METHOD containsNo
VAR_INPUT
	(* current string to check *)
	stringToCheck	:ANY_STRING;
	(* string that must not be found in ``stringToCheck`` *)
	searchString	:ANY_STRING;
	(* ``TRUE`` means ignore cases; ``FALSE`` means cases must be equal too *)
	ignoreCases		:BOOL;
	(* message if the assertion is false *)
	message			:AssertMessage;
END_VAR
IF (stringToCheck.TypeClass <> searchString.TypeClass) THEN
	THIS^.assertionWasWrong(message, THIS^.getDebugInfo('containsNo'));
	RETURN;
END_IF

IF (stringToCheck.TypeClass = __SYSTEM.TYPE_CLASS.TYPE_STRING) THEN
	THIS^.win1252Assertions.win1252ContainsNo(
		stringToCheck := stringToCheck.pValue,
		searchString := searchString.pValue,
		ignoreCases := ignoreCases,
		message := message
	);
ELSIF (stringToCheck.TypeClass = __SYSTEM.TYPE_CLASS.TYPE_WSTRING) THEN
	THIS^.utf16Assertions.utf16ContainsNo(
		stringToCheck := stringToCheck.pValue,
		searchString := searchString.pValue,
		ignoreCases := ignoreCases,
		message := message
	);
END_IF
END_METHOD

(*

short summary
=================
This assertion method checks if the current string ``stringToCheck`` ends with ``end``

.. attention:: 
	All strings are handled as null terminated byte/word streams.
	For windows-1252 is end of the string 16#00
	For UTF-16 is end of the string 16#00_00

.. attention:: 
	Method uses ``ANY_STRING`` and for this it's not possible
	to use literals/constants, because for ``ANY`` types the
	compiler generates``__SYSTEM.AnyType`` and 
	``__SYSTEM.AnyType`` contains a pointer  

.. attention:: 
	end of the string is **ALWAYS** the right side of the string 
	even for writings which written from right to left like Hebrew or Arabic

.. <legal notes>

legal notes
=================
| SPDX-FileCopyrightText: © 2022 ekvip automation GmbH <info@ekvip.de>
| SPDX-License-Identifier: Apache-2.0
| For details check: Apache-2.0_

.. _Apache-2.0: https://www.apache.org/licenses/LICENSE-2.0

.. </legal notes>

parameters
=================

*)

METHOD endsWith
VAR_INPUT
	(* current string to check *)
	stringToCheck	:ANY_STRING;
	(* expected end of ``stringToCheck`` *)
	end				:ANY_STRING;
	(* ``TRUE`` means ignore cases; ``FALSE`` means cases must be equal too *)
	ignoreCases		:BOOL;
	(* ``TRUE`` means truncation of spaces on the right side of ``stringToCheck``*)
	trim			:BOOL;
	(* message if the assertion is false *)
	message			:AssertMessage;
END_VAR
IF (stringToCheck.TypeClass <> end.TypeClass) THEN
	THIS^.assertionWasWrong(message, THIS^.getDebugInfo('endsWith'));
	RETURN;
END_IF

IF (stringToCheck.TypeClass = __SYSTEM.TYPE_CLASS.TYPE_STRING) THEN
	THIS^.win1252Assertions.win1252EndsWith(
		stringToCheck := stringToCheck.pValue,
		end := end.pValue,
		ignoreCases := ignoreCases,
		trim := trim,
		message := message
	);
ELSIF (stringToCheck.TypeClass = __SYSTEM.TYPE_CLASS.TYPE_WSTRING) THEN
	THIS^.utf16Assertions.utf16EndsWith(
		stringToCheck := stringToCheck.pValue,
		end := end.pValue,
		ignoreCases := ignoreCases,
		trim := trim,
		message := message
	);	
END_IF
END_METHOD

(*

short summary
=================
This assertion method checks if the current string ``stringToCheck`` is empty

.. attention:: 
	All strings are handled as null terminated byte/word streams.
	For windows-1252 is end of the string 16#00
	For UTF-16 is end of the string 16#00_00

.. attention:: 
	Method uses ``ANY_STRING`` and for this it's not possible
	to use literals/constants, because for ``ANY`` types the
	compiler generates``__SYSTEM.AnyType`` and 
	``__SYSTEM.AnyType`` contains a pointer  

.. <legal notes>

legal notes
=================
| SPDX-FileCopyrightText: © 2022 ekvip automation GmbH <info@ekvip.de>
| SPDX-License-Identifier: Apache-2.0
| For details check: Apache-2.0_

.. _Apache-2.0: https://www.apache.org/licenses/LICENSE-2.0

.. </legal notes>

parameters
=================

*)

METHOD isEmpty
VAR_INPUT
	(* current string to check *)
	stringToCheck	:ANY_STRING;
	(* message if the assertion is false *)
	message			:AssertMessage;
END_VAR
VAR CONSTANT
	(* strings are null terminated *)
	END_OF_WINDOWS_1252_STRING	:BYTE := 16#00;
	(* strings are null terminated *)
	END_OF_UTF16_STRING	:WORD := 16#0000;
END_VAR
IF (stringToCheck.TypeClass = __SYSTEM.TYPE_CLASS.TYPE_STRING) THEN
	IF (stringToCheck.pValue^ <> END_OF_WINDOWS_1252_STRING) THEN
		THIS^.assertionWasWrong(message, THIS^.getDebugInfo('isEmpty'));
	END_IF
ELSIF (stringToCheck.TypeClass = __SYSTEM.TYPE_CLASS.TYPE_WSTRING) THEN
	IF (stringToCheck.pValue^ <> END_OF_UTF16_STRING) THEN
		THIS^.assertionWasWrong(message, THIS^.getDebugInfo('isEmpty'));
	END_IF
END_IF
END_METHOD

(*

short summary
=================
This assertion method checks if the current string ``stringToCheck`` is equal to ``expected``

.. attention:: 
	All strings are handled as null terminated byte/word streams.
	For windows-1252 is end of the string 16#00
	For UTF-16 is end of the string 16#00_00

.. attention:: 
	Method uses ``ANY_STRING`` and for this it's not possible
	to use literals/constants, because for ``ANY`` types the
	compiler generates``__SYSTEM.AnyType`` and 
	``__SYSTEM.AnyType`` contains a pointer  

.. <legal notes>

legal notes
=================
| SPDX-FileCopyrightText: © 2022 ekvip automation GmbH <info@ekvip.de>
| SPDX-License-Identifier: Apache-2.0
| For details check: Apache-2.0_

.. _Apache-2.0: https://www.apache.org/licenses/LICENSE-2.0

.. </legal notes>

parameters
=================

*)

METHOD isEqualTo
VAR_INPUT
	(* current string to check *)
	stringToCheck	:ANY_STRING;
	(* ``stringToCheck`` must be equal to expected *)
	expected		:ANY_STRING;
	(* ``TRUE`` means ignore cases; ``FALSE`` means cases must be equal too *)
	ignoreCases		:BOOL;
	(* message if the assertion is false *)
	message			:AssertMessage;
END_VAR
IF (stringToCheck.TypeClass <> expected.TypeClass) THEN
	THIS^.assertionWasWrong(message, THIS^.getDebugInfo('isEqualTo'));
	RETURN;
END_IF

IF (stringToCheck.TypeClass = __SYSTEM.TYPE_CLASS.TYPE_STRING) THEN
	THIS^.win1252Assertions.win1252IsEqualTo(
		stringToCheck := stringToCheck.pValue,
		expected := expected.pValue,
		ignoreCases := ignoreCases,
		message := message
	);
ELSIF (stringToCheck.TypeClass = __SYSTEM.TYPE_CLASS.TYPE_WSTRING) THEN
	THIS^.utf16Assertions.utf16IsEqualTo(
		stringToCheck := stringToCheck.pValue,
		expected := expected.pValue,
		ignoreCases := ignoreCases,
		message := message
	);	
END_IF
END_METHOD

(*

short summary
=================
This assertion method checks if the current string ``stringToCheck`` is not empty

.. attention:: 
	All strings are handled as null terminated byte/word streams.
	For windows-1252 is end of the string 16#00
	For UTF-16 is end of the string 16#00_00

.. attention:: 
	Method uses ``ANY_STRING`` and for this it's not possible
	to use literals/constants, because for ``ANY`` types the
	compiler generates``__SYSTEM.AnyType`` and 
	``__SYSTEM.AnyType`` contains a pointer  

.. <legal notes>

legal notes
=================
| SPDX-FileCopyrightText: © 2022 ekvip automation GmbH <info@ekvip.de>
| SPDX-License-Identifier: Apache-2.0
| For details check: Apache-2.0_

.. _Apache-2.0: https://www.apache.org/licenses/LICENSE-2.0

.. </legal notes>

parameters
=================

*)

METHOD isNotEmpty
VAR_INPUT
	(* current string to check *)
	stringToCheck	:ANY_STRING;
	(* message if the assertion is false *)
	message			:AssertMessage;
END_VAR
VAR CONSTANT
	(* strings are null terminated *)
	END_OF_WINDOWS_1252_STRING	:BYTE := 16#00;
	(* strings are null terminated *)
	END_OF_UTF16_STRING	:WORD := 16#0000;
END_VAR
IF (stringToCheck.TypeClass = __SYSTEM.TYPE_CLASS.TYPE_STRING) THEN
	IF (stringToCheck.pValue^ = END_OF_WINDOWS_1252_STRING) THEN
		THIS^.assertionWasWrong(message, THIS^.getDebugInfo('isNotEmpty'));
	END_IF
ELSIF (stringToCheck.TypeClass = __SYSTEM.TYPE_CLASS.TYPE_WSTRING) THEN
	IF (stringToCheck.pValue^ = END_OF_UTF16_STRING) THEN
		THIS^.assertionWasWrong(message, THIS^.getDebugInfo('isNotEmpty'));
	END_IF
END_IF
END_METHOD

(*

short summary
=================
This assertion method checks if the current string ``stringToCheck`` is not equal to ``unexpected``

.. attention:: 
	All strings are handled as null terminated byte/word streams.
	For windows-1252 is end of the string 16#00
	For UTF-16 is end of the string 16#00_00

.. attention:: 
	Method uses ``ANY_STRING`` and for this it's not possible
	to use literals/constants, because for ``ANY`` types the
	compiler generates``__SYSTEM.AnyType`` and 
	``__SYSTEM.AnyType`` contains a pointer  

.. <legal notes>

legal notes
=================
| SPDX-FileCopyrightText: © 2022 ekvip automation GmbH <info@ekvip.de>
| SPDX-License-Identifier: Apache-2.0
| For details check: Apache-2.0_

.. _Apache-2.0: https://www.apache.org/licenses/LICENSE-2.0

.. </legal notes>

parameters
=================

*)

METHOD isNotEqualTo
VAR_INPUT
	(* current string to check *)
	stringToCheck	:ANY_STRING;
	(* ``stringToCheck`` must be not equal to expected *)
	unexpected		:ANY_STRING;
	(* ``TRUE`` means ignore cases; ``FALSE`` means cases must be equal too *)
	ignoreCases		:BOOL;
	(* message if the assertion is false *)
	message			:AssertMessage;
END_VAR
IF (stringToCheck.TypeClass <> unexpected.TypeClass) THEN
	RETURN;
END_IF

IF (stringToCheck.TypeClass = __SYSTEM.TYPE_CLASS.TYPE_STRING) THEN
	THIS^.win1252Assertions.win1252IsNotEqualTo(
		stringToCheck := stringToCheck.pValue,
		unexpected := unexpected.pValue,
		ignoreCases := ignoreCases,
		message := message
	);
ELSIF (stringToCheck.TypeClass = __SYSTEM.TYPE_CLASS.TYPE_WSTRING) THEN
	THIS^.utf16Assertions.utf16IsNotEqualTo(
		stringToCheck := stringToCheck.pValue,
		unexpected := unexpected.pValue,
		ignoreCases := ignoreCases,
		message := message
	);	
END_IF
END_METHOD

(*

short summary
=================
This assertion method checks if the current string ``stringToCheck`` is length
is between ``minLenght`` and ``maxLenght``

.. attention:: 
	All strings are handled as null terminated byte/word streams.
	For windows-1252 is end of the string 16#00
	For UTF-16 is end of the string 16#00_00

.. attention:: 
	Method uses ``ANY_STRING`` and for this it's not possible
	to use literals/constants, because for ``ANY`` types the
	compiler generates``__SYSTEM.AnyType`` and 
	``__SYSTEM.AnyType`` contains a pointer  

.. <legal notes>

legal notes
=================
| SPDX-FileCopyrightText: © 2022 ekvip automation GmbH <info@ekvip.de>
| SPDX-License-Identifier: Apache-2.0
| For details check: Apache-2.0_

.. _Apache-2.0: https://www.apache.org/licenses/LICENSE-2.0

.. </legal notes>

parameters
=================

*)

METHOD lenghtIsBetween
VAR_INPUT
	(* current string to check *)
	stringToCheck	:ANY_STRING;
	(* lower limit of the string length *)
	minLenght		:UDINT;
	(* upper limit of the string length *)
	maxLenght		:UDINT;
	(* message if the assertion is false *)
	message			:AssertMessage;
END_VAR
IF (stringToCheck.TypeClass = __SYSTEM.TYPE_CLASS.TYPE_STRING) THEN
	THIS^.win1252Assertions.win1252LengthIsBetween(
		stringToCheck	:= stringToCheck.pValue,
		minLenght		:= minLenght,
		maxLenght		:= maxLenght,
		message			:= message
	);
ELSIF (stringToCheck.TypeClass = __SYSTEM.TYPE_CLASS.TYPE_WSTRING) THEN
	THIS^.utf16Assertions.utf16LengthIsBetween(
		stringToCheck	:= stringToCheck.pValue,
		minLenght		:= minLenght,
		maxLenght		:= maxLenght,
		message			:= message
	);	
END_IF
END_METHOD

(*

short summary
=================
This assertion method checks if the current string ``stringToCheck`` is length
is equal to ``expectedLength``

.. attention:: 
	All strings are handled as null terminated byte/word streams.
	For windows-1252 is end of the string 16#00
	For UTF-16 is end of the string 16#00_00

.. attention:: 
	Method uses ``ANY_STRING`` and for this it's not possible
	to use literals/constants, because for ``ANY`` types the
	compiler generates``__SYSTEM.AnyType`` and 
	``__SYSTEM.AnyType`` contains a pointer  

.. <legal notes>

legal notes
=================
| SPDX-FileCopyrightText: © 2022 ekvip automation GmbH <info@ekvip.de>
| SPDX-License-Identifier: Apache-2.0
| For details check: Apache-2.0_

.. _Apache-2.0: https://www.apache.org/licenses/LICENSE-2.0

.. </legal notes>

parameters
=================

*)

METHOD lenghtIsExact
VAR_INPUT
	(* current string to check *)
	stringToCheck	:ANY_STRING;
	(* expected length of ``stringToCheck`` *)
	expectedLength	:UDINT;
	(* message if the assertion is false *)
	message			:AssertMessage;
END_VAR
IF (stringToCheck.TypeClass = __SYSTEM.TYPE_CLASS.TYPE_STRING) THEN
	THIS^.win1252Assertions.win1252LenghtIsExact(
		stringToCheck	:= stringToCheck.pValue,
		expectedLength	:= expectedLength,
		message			:= message
	);
ELSIF (stringToCheck.TypeClass = __SYSTEM.TYPE_CLASS.TYPE_WSTRING) THEN
	THIS^.utf16Assertions.utf16LenghtIsExact(
		stringToCheck	:= stringToCheck.pValue,
		expectedLength	:= expectedLength,
		message			:= message
	);	
END_IF
END_METHOD

(*

short summary
=================
This assertion method checks if the current string ``stringToCheck`` is length
is equal or less than to ``maxLength``

.. attention:: 
	All strings are handled as null terminated byte/word streams.
	For windows-1252 is end of the string 16#00
	For UTF-16 is end of the string 16#00_00

.. attention:: 
	Method uses ``ANY_STRING`` and for this it's not possible
	to use literals/constants, because for ``ANY`` types the
	compiler generates``__SYSTEM.AnyType`` and 
	``__SYSTEM.AnyType`` contains a pointer  

.. <legal notes>

legal notes
=================
| SPDX-FileCopyrightText: © 2022 ekvip automation GmbH <info@ekvip.de>
| SPDX-License-Identifier: Apache-2.0
| For details check: Apache-2.0_

.. _Apache-2.0: https://www.apache.org/licenses/LICENSE-2.0

.. </legal notes>

parameters
=================

*)

METHOD lenghtIsMax
VAR_INPUT
	(* current string to check *)
	stringToCheck	:ANY_STRING;
	(* upper limit of the length of ``stringToCheck`` *)
	maxLength		:UDINT;
	(* message if the assertion is false *)
	message			:AssertMessage;
END_VAR
IF (stringToCheck.TypeClass = __SYSTEM.TYPE_CLASS.TYPE_STRING) THEN
	THIS^.win1252Assertions.win1252LenghtIsMax(
		stringToCheck	:= stringToCheck.pValue,
		maxLength		:= maxLength,
		message			:= message
	);
ELSIF (stringToCheck.TypeClass = __SYSTEM.TYPE_CLASS.TYPE_WSTRING) THEN
	THIS^.utf16Assertions.utf16LenghtIsMax(
		stringToCheck	:= stringToCheck.pValue,
		maxLength		:= maxLength,
		message			:= message
	);	
END_IF
END_METHOD

(*

short summary
=================
This assertion method checks if the current string ``stringToCheck`` is length
is equal or grater than to ``minLength``

.. attention:: 
	All strings are handled as null terminated byte/word streams.
	For windows-1252 is end of the string 16#00
	For UTF-16 is end of the string 16#00_00

.. attention:: 
	Method uses ``ANY_STRING`` and for this it's not possible
	to use literals/constants, because for ``ANY`` types the
	compiler generates``__SYSTEM.AnyType`` and 
	``__SYSTEM.AnyType`` contains a pointer  

.. <legal notes>

legal notes
=================
| SPDX-FileCopyrightText: © 2022 ekvip automation GmbH <info@ekvip.de>
| SPDX-License-Identifier: Apache-2.0
| For details check: Apache-2.0_

.. _Apache-2.0: https://www.apache.org/licenses/LICENSE-2.0

.. </legal notes>

parameters
=================

*)

METHOD lenghtIsMin
VAR_INPUT
	(* current string to check *)
	stringToCheck	:ANY_STRING;
	(* lower limit of the length of ``stringToCheck`` *)
	minLength		:UDINT;
	(* message if the assertion is false *)
	message			:AssertMessage;
END_VAR
IF (stringToCheck.TypeClass = __SYSTEM.TYPE_CLASS.TYPE_STRING) THEN
	THIS^.win1252Assertions.win1252LenghtIsMin(
		stringToCheck	:= stringToCheck.pValue,
		minLength		:= minLength,
		message			:= message
	);
ELSIF (stringToCheck.TypeClass = __SYSTEM.TYPE_CLASS.TYPE_WSTRING) THEN
	THIS^.utf16Assertions.utf16LenghtIsMin(
		stringToCheck	:= stringToCheck.pValue,
		minLength		:= minLength,
		message			:= message
	);
END_IF
END_METHOD

(*

short summary
=================
This methods is the setter for the callback class if an assertion was false

.. <legal notes>

legal notes
=================
| SPDX-FileCopyrightText: © 2022 ekvip automation GmbH <info@ekvip.de>
| SPDX-License-Identifier: Apache-2.0
| For details check: Apache-2.0_

.. _Apache-2.0: https://www.apache.org/licenses/LICENSE-2.0

.. </legal notes>

parameters
=================

*)

METHOD setCallBack
VAR_INPUT
	(* the class that must be informed if an assertion is false *)
	callBack	:IAssertCallback;  
END_VAR
SUPER^.setCallBack(callBack);
THIS^.win1252Assertions.setCallBack(callBack);
THIS^.utf16Assertions.setCallBack(callBack);
END_METHOD

(*

short summary
=================
This assertion method checks if the current string ``stringToCheck`` starts with ``start``

.. attention:: 
	All strings are handled as null terminated byte/word streams.
	For windows-1252 is end of the string 16#00
	For UTF-16 is end of the string 16#00_00

.. attention:: 
	Method uses ``ANY_STRING`` and for this it's not possible
	to use literals/constants, because for ``ANY`` types the
	compiler generates``__SYSTEM.AnyType`` and 
	``__SYSTEM.AnyType`` contains a pointer  

.. attention:: 
	start of the string is **ALWAYS** the left side of the string 
	even for writings which written from right to left like Hebrew or Arabic

.. <legal notes>

legal notes
=================
| SPDX-FileCopyrightText: © 2022 ekvip automation GmbH <info@ekvip.de>
| SPDX-License-Identifier: Apache-2.0
| For details check: Apache-2.0_

.. _Apache-2.0: https://www.apache.org/licenses/LICENSE-2.0

.. </legal notes>

parameters
=================

*)

METHOD startsWith
VAR_INPUT
	(* current string to check *)
	stringToCheck	:ANY_STRING;
	(* expected start of ``stringToCheck`` *)
	start			:ANY_STRING;
	(* ``TRUE`` means ignore cases; ``FALSE`` means cases must be equal too *)
	ignoreCases		:BOOL;
	(* ``TRUE`` means truncation of spaces on the left side of ``stringToCheck``*)
	trim			:BOOL;
	(* message if the assertion is false *)
	message			:AssertMessage;
END_VAR
IF (stringToCheck.TypeClass <> start.TypeClass) THEN
	THIS^.assertionWasWrong(message, THIS^.getDebugInfo('startsWith'));
	RETURN;
END_IF

IF (stringToCheck.TypeClass = __SYSTEM.TYPE_CLASS.TYPE_STRING) THEN
	THIS^.win1252Assertions.win1252StartsWith(
		stringToCheck := stringToCheck.pValue,
		start := start.pValue,
		ignoreCases := ignoreCases,
		trim := trim,
		message := message
	);
ELSIF (stringToCheck.TypeClass = __SYSTEM.TYPE_CLASS.TYPE_WSTRING) THEN
	THIS^.utf16Assertions.utf16StartsWith(
		stringToCheck := stringToCheck.pValue,
		start := start.pValue,
		ignoreCases := ignoreCases,
		trim := trim,
		message := message
	);
END_IF
END_METHOD

END_FUNCTION_BLOCK

// ---- Assertor/Assertions/TimeAssertions/classes/TimeAssertions.TcPOU
(*

short summary
=================
This class implements the interface :ref:`ITimeAssertions`.
It provides assertions for time data types
For ``LTIME`` assertions use :ref:`TimeAssertions.long`.
For ``TIME`` assertions use :ref:`TimeAssertions.simple`.


.. <legal notes>

legal notes
=================
| SPDX-FileCopyrightText: © 2022 ekvip automation GmbH <info@ekvip.de>
| SPDX-License-Identifier: Apache-2.0
| For details check: Apache-2.0_

.. _Apache-2.0: https://www.apache.org/licenses/LICENSE-2.0

.. </legal notes>

methods and properties
=========================

*)

{attribute 'reflection'}
FUNCTION_BLOCK INTERNAL TimeAssertions EXTENDS CNM_AbstractObject.Object IMPLEMENTS ITimeAssertions, IAssertCallBackSetter
VAR
	(* class to handle TIME assertions *)
	simpleTimeAssertions	:SimpleTimeAssertions();
	(* class to handle LTIME assertions *)
	longTimeAssertions		:LongTimeAssertions();
END_VAR

(*

short summary
=================
This abstract property returns the class name of the concrete object, 
It's for debugging purpose

.. <legal notes>

legal notes
=================
| SPDX-FileCopyrightText: © 2022 ekvip automation GmbH <info@ekvip.de>
| SPDX-License-Identifier: Apache-2.0
| For details check: Apache-2.0_

.. _Apache-2.0: https://www.apache.org/licenses/LICENSE-2.0

.. </legal notes>

*)

PROPERTY className :ClassName
GET
className := 'CNM_AssertionInterfaceLib.TimeAssertions';
END_GET
END_PROPERTY

(*

short summary
=================
Returns an interface (:ref:`I64BitTimeAssertions`)
with assert statements for 64 bit times 

.. <legal notes>

legal notes
=================
| SPDX-FileCopyrightText: © 2022 ekvip automation GmbH <info@ekvip.de>
| SPDX-License-Identifier: Apache-2.0
| For details check: Apache-2.0_

.. _Apache-2.0: https://www.apache.org/licenses/LICENSE-2.0

.. </legal notes>

*)

PROPERTY long :I64BitTimeAssertions
GET
long := THIS^.longTimeAssertions;
END_GET
END_PROPERTY

(*

short summary
=================
This methods is the setter for the callback class if an assertion was false

.. <legal notes>

legal notes
=================
| SPDX-FileCopyrightText: © 2022 ekvip automation GmbH <info@ekvip.de>
| SPDX-License-Identifier: Apache-2.0
| For details check: Apache-2.0_

.. _Apache-2.0: https://www.apache.org/licenses/LICENSE-2.0

.. </legal notes>

parameters
=================

*)

METHOD setCallBack
VAR_INPUT
	(* the class that must be informed if an assertion is false *)
	callBack	:IAssertCallback;  
END_VAR
THIS^.simpleTimeAssertions.setCallBack(callBack);
THIS^.longTimeAssertions.setCallBack(callBack);
END_METHOD

(*

short summary
=================
Returns an interface (:ref:`I32BitTimeAssertions`)
with assert statements for 32 bit times 

.. <legal notes>

legal notes
=================
| SPDX-FileCopyrightText: © 2022 ekvip automation GmbH <info@ekvip.de>
| SPDX-License-Identifier: Apache-2.0
| For details check: Apache-2.0_

.. _Apache-2.0: https://www.apache.org/licenses/LICENSE-2.0

.. </legal notes>

*)

PROPERTY simple :I32BitTimeAssertions
GET
simple := THIS^.simpleTimeAssertions;
END_GET
END_PROPERTY

END_FUNCTION_BLOCK

// ---- Assertor/Assertions/TimeAssertions/Time/classes/SimpleTimeAssertions.TcPOU
(*

short summary
=================
This class implements the interface :ref:`I32BitTimeAssertions`. 
It contains the assert statements for the data type ``TIME``

.. <legal notes>

legal notes
=================
| SPDX-FileCopyrightText: © 2022 ekvip automation GmbH <info@ekvip.de>
| SPDX-License-Identifier: Apache-2.0
| For details check: Apache-2.0_

.. _Apache-2.0: https://www.apache.org/licenses/LICENSE-2.0

.. </legal notes>

methods and properties
=========================

*)

{attribute 'reflection'}
FUNCTION_BLOCK INTERNAL SimpleTimeAssertions EXTENDS AbstactAssertion IMPLEMENTS I32BitTimeAssertions
VAR CONSTANT
	(* maximum value for the data type ``TIME`` *)
	MAX_TIME	:TIME := TO_TIME(16#FF_FF_FF_FF);
END_VAR

(*

short summary
=================
This abstract property returns the class name of the concrete object, 
It's for debugging purpose

.. <legal notes>

legal notes
=================
| SPDX-FileCopyrightText: © 2022 ekvip automation GmbH <info@ekvip.de>
| SPDX-License-Identifier: Apache-2.0
| For details check: Apache-2.0_

.. _Apache-2.0: https://www.apache.org/licenses/LICENSE-2.0

.. </legal notes>

*)

PROPERTY className :ClassName
GET
className := 'CNM_AssertionInterfaceLib.SimplyTimeAssertions';
END_GET
END_PROPERTY

(*

short summary
=================
This method returns the passed time since the timestamp was created

.. <legal notes>

legal notes
=================
| SPDX-FileCopyrightText: © 2022 ekvip automation GmbH <info@ekvip.de>
| SPDX-License-Identifier: Apache-2.0
| For details check: Apache-2.0_

.. _Apache-2.0: https://www.apache.org/licenses/LICENSE-2.0

.. </legal notes>

parameters
=================
:return: passed time since ``startTime``

*)

METHOD PROTECTED getTimePassed :TIME
VAR_INPUT
	(* timestamp start *)
	startTime	:TIME;
END_VAR
VAR
	(* current time to calculate the passed time *)
	currentTime	:TIME;
END_VAR
currentTime := TIME();
IF (currentTime > startTime) THEN
	getTimePassed := (currentTime - startTime);
ELSE
	getTimePassed := ((THIS^.MAX_TIME - startTime) + currentTime);
END_IF
END_METHOD

(*

short summary
=================
This assertion method checks whether time has elapsed since the timestamp time

.. <legal notes>

legal notes
=================
| SPDX-FileCopyrightText: © 2022 ekvip automation GmbH <info@ekvip.de>
| SPDX-License-Identifier: Apache-2.0
| For details check: Apache-2.0_

.. _Apache-2.0: https://www.apache.org/licenses/LICENSE-2.0

.. </legal notes>

parameters
=================

*)

METHOD timeHasExpired
VAR_INPUT
	(* start time you get it with ``TIME()`` *)
	timestamp		:TIME;
	(* timeout like ``t#300ms`` *)
	expiringTime	:TIME;
	(* message if the assertion is false *)
	message			:AssertMessage;
END_VAR
VAR
	(* measured passed time *)
	passedTime		:TIME;
END_VAR
passedTime := THIS^.getTimePassed(timestamp);
IF (passedTime < expiringTime) THEN
	THIS^.assertionWasWrong(
		message			:= message,
		additionalText	:= THIS^.getDebugInfo('timeHasExpired')
	);	
END_IF
END_METHOD

(*

short summary
=================
This assertion method checks that the time since the timestamp time has not yet elapsed

.. <legal notes>

legal notes
=================
| SPDX-FileCopyrightText: © 2022 ekvip automation GmbH <info@ekvip.de>
| SPDX-License-Identifier: Apache-2.0
| For details check: Apache-2.0_

.. _Apache-2.0: https://www.apache.org/licenses/LICENSE-2.0

.. </legal notes>

parameters
=================

*)

METHOD timeHasNotExpired
VAR_INPUT
	(* start time you get it with ``TIME()`` *)
	timestamp		:TIME;
	(* timeout like ``t#300ms`` *)
	expiringTime	:TIME;
	(* message if the assertion is false *)
	message			:AssertMessage;
END_VAR
VAR
	(* measured passed time *)
	passedTime		:TIME;
END_VAR
passedTime := THIS^.getTimePassed(timestamp);
IF (passedTime >= expiringTime) THEN
	THIS^.assertionWasWrong(
		message			:= message,
		additionalText	:= THIS^.getDebugInfo('timeHasNotExpired')
	);	
END_IF
END_METHOD

(*

short summary
=================
This assertion method checks if the current value is equal to the expected value

.. <legal notes>

legal notes
=================
| SPDX-FileCopyrightText: © 2022 ekvip automation GmbH <info@ekvip.de>
| SPDX-License-Identifier: Apache-2.0
| For details check: Apache-2.0_

.. _Apache-2.0: https://www.apache.org/licenses/LICENSE-2.0

.. </legal notes>

parameters
=================

*)

METHOD valueIsEqualTo
VAR_INPUT
	(* current value to check *)
	currentValue	:TIME;
	(* expected value to compare *)
	expectedValue	:TIME;
	(* message if the assertion is false *)
	message			:AssertMessage;
END_VAR
IF (currentValue <> expectedValue) THEN
	THIS^.assertionWasWrong(
		message			:= message,
		additionalText	:= THIS^.getDebugInfo('valueIsEqualTo')
	);	
END_IF
END_METHOD

(*

short summary
=================
This assertion method checks if the current value is greater than the less value

.. <legal notes>

legal notes
=================
| SPDX-FileCopyrightText: © 2022 ekvip automation GmbH <info@ekvip.de>
| SPDX-License-Identifier: Apache-2.0
| For details check: Apache-2.0_

.. _Apache-2.0: https://www.apache.org/licenses/LICENSE-2.0

.. </legal notes>

parameters
=================

*)

METHOD valueIsGreaterThan
VAR_INPUT
	(* current value to check *)
	currentValue	:TIME;
	(* less than lower limit *)
	lessValue		:TIME;
	(* message if the assertion is false *)
	message			:AssertMessage;
END_VAR
IF (currentValue <= lessValue) THEN
	THIS^.assertionWasWrong(
		message			:= message,
		additionalText	:= THIS^.getDebugInfo('valueIsGreaterThan')
	);	
END_IF
END_METHOD

(*

short summary
=================
This assertion method checks if the current value is inside a limit

.. attention:: 
	limits are included: ``valueIsInRangeOf(t#3ms,t#3ms ,t#3ms)`` is a true assertion

.. <legal notes>

legal notes
=================
| SPDX-FileCopyrightText: © 2022 ekvip automation GmbH <info@ekvip.de>
| SPDX-License-Identifier: Apache-2.0
| For details check: Apache-2.0_

.. _Apache-2.0: https://www.apache.org/licenses/LICENSE-2.0

.. </legal notes>

parameters
=================

*)

METHOD valueIsInRangeOf
VAR_INPUT
	(* lower limit for the current value *)
	lowerLimit		:TIME;
	(* current value to check *)
	currentValue	:TIME;
	(* upper limit for the current value *)
	upperLimit		:TIME;
	(* message if the assertion is false *)
	message			:AssertMessage;
END_VAR
IF ((currentValue < lowerLimit) OR (currentValue > upperLimit)) THEN
	THIS^.assertionWasWrong(
		message			:= message,
		additionalText	:= THIS^.getDebugInfo('valueIsInRangeOf')
	);	
END_IF
END_METHOD

(*

short summary
=================
This assertion method checks if the current value is less than the greater value

.. <legal notes>

legal notes
=================
| SPDX-FileCopyrightText: © 2022 ekvip automation GmbH <info@ekvip.de>
| SPDX-License-Identifier: Apache-2.0
| For details check: Apache-2.0_

.. _Apache-2.0: https://www.apache.org/licenses/LICENSE-2.0

.. </legal notes>

parameters
=================

*)

METHOD valueIsLessThan
VAR_INPUT
	(* current value to check *)
	currentValue	:TIME;
	(* greater than upper limit *)
	greaterValue	:TIME;
	(* message if the assertion is false *)
	message			:AssertMessage;
END_VAR
IF (currentValue >= greaterValue) THEN
	THIS^.assertionWasWrong(
		message			:= message,
		additionalText	:= THIS^.getDebugInfo('valueIsLessThan')
	);	
END_IF
END_METHOD

(*

short summary
=================
This assertion method checks if the current value is less than or equal to the maximum value

.. <legal notes>

legal notes
=================
| SPDX-FileCopyrightText: © 2022 ekvip automation GmbH <info@ekvip.de>
| SPDX-License-Identifier: Apache-2.0
| For details check: Apache-2.0_

.. _Apache-2.0: https://www.apache.org/licenses/LICENSE-2.0

.. </legal notes>

parameters
=================

*)

METHOD valueIsMax
VAR_INPUT
	(* current value to check *)
	currentValue	:TIME;
	(* upper limit for the current value *)
	maximumValue	:TIME;
	(* message if the assertion is false *)
	message			:AssertMessage;
END_VAR
IF (currentValue > maximumValue) THEN
	THIS^.assertionWasWrong(
		message			:= message,
		additionalText	:= THIS^.getDebugInfo('valueIsMax')
	);	
END_IF
END_METHOD

(*

short summary
=================
This assertion method checks if the current value is greater than or equal to the minimum value

.. <legal notes>

legal notes
=================
| SPDX-FileCopyrightText: © 2022 ekvip automation GmbH <info@ekvip.de>
| SPDX-License-Identifier: Apache-2.0
| For details check: Apache-2.0_

.. _Apache-2.0: https://www.apache.org/licenses/LICENSE-2.0

.. </legal notes>

parameters
=================

*)

METHOD valueIsMin
VAR_INPUT
	(* current value to check *)
	currentValue	:TIME;
	(* lower limit for the current value *)
	minimumValue	:TIME;
	(* message if the assertion is false *)
	message			:AssertMessage;
END_VAR
IF (currentValue < minimumValue) THEN
	THIS^.assertionWasWrong(
		message			:= message,
		additionalText	:= THIS^.getDebugInfo('valueIsMin')
	);	
END_IF
END_METHOD

(*

short summary
=================
This assertion method checks if the current value is not equal to the unexpected value

.. <legal notes>

legal notes
=================
| SPDX-FileCopyrightText: © 2022 ekvip automation GmbH <info@ekvip.de>
| SPDX-License-Identifier: Apache-2.0
| For details check: Apache-2.0_

.. _Apache-2.0: https://www.apache.org/licenses/LICENSE-2.0

.. </legal notes>

parameters
=================

*)

METHOD valueIsNotEqualTo
VAR_INPUT
	(* current value to check *)
	currentValue	:TIME;
	(* unexpected value to compare *)
	unexpectedValue	:TIME;
	(* message if the assertion is false *)
	message			:AssertMessage;
END_VAR
IF (currentValue = unexpectedValue) THEN
	THIS^.assertionWasWrong(
		message			:= message,
		additionalText	:= THIS^.getDebugInfo('valueIsNotEqualTo')
	);	
END_IF
END_METHOD

END_FUNCTION_BLOCK

// ---- Assertor/Assertions/TimeAssertions/LTime/classes/LongTimeAssertions.TcPOU
(*

short summary
=================
This class implements the interface :ref:`I64BitTimeAssertions`. 
It provides the assert statements for the data type ``LTIME``

.. <legal notes>

legal notes
=================
| SPDX-FileCopyrightText: © 2022 ekvip automation GmbH <info@ekvip.de>
| SPDX-License-Identifier: Apache-2.0
| For details check: Apache-2.0_

.. _Apache-2.0: https://www.apache.org/licenses/LICENSE-2.0

.. </legal notes>

methods and properties
=========================

*)

{attribute 'reflection'}
FUNCTION_BLOCK INTERNAL LongTimeAssertions EXTENDS AbstactAssertion IMPLEMENTS I64BitTimeAssertions
VAR CONSTANT
	(* maximum value for the data type ``LTIME`` *)
	MAX_TIME	:LTIME := TO_LTIME(16#FFFF_FFFF_FFFF_FFFF);
END_VAR

(*

short summary
=================
This abstract property returns the class name of the concrete object, 
It's for debugging purpose

.. <legal notes>

legal notes
=================
| SPDX-FileCopyrightText: © 2022 ekvip automation GmbH <info@ekvip.de>
| SPDX-License-Identifier: Apache-2.0
| For details check: Apache-2.0_

.. _Apache-2.0: https://www.apache.org/licenses/LICENSE-2.0

.. </legal notes>

*)

PROPERTY className :ClassName
GET
className := 'CNM_AssertionInterfaceLib.LongTimeAssertions';
END_GET
END_PROPERTY

(*

short summary
=================
This method returns the passed time since the timestamp was created

.. <legal notes>

legal notes
=================
| SPDX-FileCopyrightText: © 2022 ekvip automation GmbH <info@ekvip.de>
| SPDX-License-Identifier: Apache-2.0
| For details check: Apache-2.0_

.. _Apache-2.0: https://www.apache.org/licenses/LICENSE-2.0

.. </legal notes>

parameters
=================
:return: passed time since ``startTime``

*)

METHOD PROTECTED getTimePassed :LTIME
VAR_INPUT
	(* timestamp start *)
	startTime	:LTIME;
END_VAR
VAR
	(* current time to calculate the passed time *)
	currentTime	:LTIME;
END_VAR
currentTime := LTIME();
IF (currentTime > startTime) THEN
	getTimePassed := (currentTime - startTime);
ELSE
	getTimePassed := ((THIS^.MAX_TIME - startTime) + currentTime);
END_IF
END_METHOD

(*

short summary
=================
This assertion method checks whether time has elapsed since the timestamp time

.. <legal notes>

legal notes
=================
| SPDX-FileCopyrightText: © 2022 ekvip automation GmbH <info@ekvip.de>
| SPDX-License-Identifier: Apache-2.0
| For details check: Apache-2.0_

.. _Apache-2.0: https://www.apache.org/licenses/LICENSE-2.0

.. </legal notes>

parameters
=================

*)

METHOD timeHasExpired
VAR_INPUT
	(* start time you get it with ``LTIME()`` *)
	timestamp		:LTIME;
	(* timeout like ``lt#300ms`` *)
	expiringTime	:LTIME;
	(* message if the assertion is false *)
	message			:AssertMessage;
END_VAR
VAR
	(* measured passed time *)
	passedTime		:LTIME;
END_VAR
passedTime := THIS^.getTimePassed(timestamp);
IF (passedTime < expiringTime) THEN
	THIS^.assertionWasWrong(
		message			:= message,
		additionalText	:= THIS^.getDebugInfo('timeHasExpired')
	);	
END_IF
END_METHOD

(*

short summary
=================
This assertion method checks that the time since the timestamp time has not yet elapsed

.. <legal notes>

legal notes
=================
| SPDX-FileCopyrightText: © 2022 ekvip automation GmbH <info@ekvip.de>
| SPDX-License-Identifier: Apache-2.0
| For details check: Apache-2.0_

.. _Apache-2.0: https://www.apache.org/licenses/LICENSE-2.0

.. </legal notes>

parameters
=================

*)

METHOD timeHasNotExpired
VAR_INPUT
	(* start time you get it with ``LTIME()`` *)
	timestamp		:LTIME;
	(* timeout like ``lt#300ms`` *)
	expiringTime	:LTIME;
	(* message if the assertion is false *)
	message			:AssertMessage;
END_VAR
VAR
	(* measured passed time *)
	passedTime		:LTIME;
END_VAR
passedTime := THIS^.getTimePassed(timestamp);
IF (passedTime >= expiringTime) THEN
	THIS^.assertionWasWrong(
		message			:= message,
		additionalText	:= THIS^.getDebugInfo('timeHasNotExpired')
	);	
END_IF
END_METHOD

(*

short summary
=================
This assertion method checks if the current value is equal to the expected value

.. <legal notes>

legal notes
=================
| SPDX-FileCopyrightText: © 2022 ekvip automation GmbH <info@ekvip.de>
| SPDX-License-Identifier: Apache-2.0
| For details check: Apache-2.0_

.. _Apache-2.0: https://www.apache.org/licenses/LICENSE-2.0

.. </legal notes>

parameters
=================

*)

METHOD valueIsEqualTo
VAR_INPUT
	(* current value to check *)
	currentValue	:LTIME;
	(* expected value to compare *)
	expectedValue	:LTIME;
	(* message if the assertion is false *)
	message	:AssertMessage;
END_VAR
IF (currentValue <> expectedValue) THEN
	THIS^.assertionWasWrong(
		message			:= message,
		additionalText	:= THIS^.getDebugInfo('valueIsEqualTo')
	);	
END_IF
END_METHOD

(*

short summary
=================
This assertion method checks if the current value is greater than the less value

.. <legal notes>

legal notes
=================
| SPDX-FileCopyrightText: © 2022 ekvip automation GmbH <info@ekvip.de>
| SPDX-License-Identifier: Apache-2.0
| For details check: Apache-2.0_

.. _Apache-2.0: https://www.apache.org/licenses/LICENSE-2.0

.. </legal notes>

parameters
=================

*)

METHOD valueIsGreaterThan
VAR_INPUT
	(* current value to check *)
	currentValue	:LTIME;
	(* less than lower limit *)
	lessValue		:LTIME;
	(* message if the assertion is false *)
	message	: AssertMessage;
END_VAR
IF (currentValue <= lessValue) THEN
	THIS^.assertionWasWrong(
		message			:= message,
		additionalText	:= THIS^.getDebugInfo('valueIsGreaterThan')
	);	
END_IF
END_METHOD

(*

short summary
=================
This assertion method checks if the current value is inside a limit

.. attention:: 
	limits are included: ``valueIsInRangeOf(t#3ms,t#3ms ,t#3ms)`` is a true assertion

.. <legal notes>

legal notes
=================
| SPDX-FileCopyrightText: © 2022 ekvip automation GmbH <info@ekvip.de>
| SPDX-License-Identifier: Apache-2.0
| For details check: Apache-2.0_

.. _Apache-2.0: https://www.apache.org/licenses/LICENSE-2.0

.. </legal notes>

parameters
=================

*)

METHOD valueIsInRangeOf
VAR_INPUT
	(* lower limit for the current value *)
	lowerLimit		:LTIME;
	(* current value to check *)
	currentValue	:LTIME;
	(* upper limit for the current value *)
	upperLimit		:LTIME;
	(* message if the assertion is false *)
	message			:AssertMessage;
END_VAR
VAR
	(* additional information for the callback function *)
	additionalText	:Tc2_System.T_MaxString;
END_VAR
IF ((currentValue < lowerLimit) OR (currentValue > upperLimit)) THEN
	THIS^.assertionWasWrong(
		message			:= message,
		additionalText	:= THIS^.getDebugInfo('valueIsInRangeOf')
	);	
END_IF
END_METHOD

(*

short summary
=================
This assertion method checks if the current value is less than the greater value

.. <legal notes>

legal notes
=================
| SPDX-FileCopyrightText: © 2022 ekvip automation GmbH <info@ekvip.de>
| SPDX-License-Identifier: Apache-2.0
| For details check: Apache-2.0_

.. _Apache-2.0: https://www.apache.org/licenses/LICENSE-2.0

.. </legal notes>

parameters
=================

*)

METHOD valueIsLessThan
VAR_INPUT
	(* current value to check *)
	currentValue	:LTIME;
	(* greater than upper limit *)
	greaterValue	:LTIME;
	(* message if the assertion is false *)
	message			:AssertMessage;
END_VAR
IF (currentValue >= greaterValue) THEN
	THIS^.assertionWasWrong(
		message			:= message,
		additionalText	:= THIS^.getDebugInfo('valueIsLessThan')
	);	
END_IF
END_METHOD

(*

short summary
=================
This assertion method checks if the current value is less than or equal to the maximum value

.. <legal notes>

legal notes
=================
| SPDX-FileCopyrightText: © 2022 ekvip automation GmbH <info@ekvip.de>
| SPDX-License-Identifier: Apache-2.0
| For details check: Apache-2.0_

.. _Apache-2.0: https://www.apache.org/licenses/LICENSE-2.0

.. </legal notes>

parameters
=================

*)

METHOD valueIsMax
VAR_INPUT
	(* current value to check *)
	currentValue	:LTIME;
	(* upper limit for the current value *)
	maximumValue	:LTIME;
	(* message if the assertion is false *)
	message			:AssertMessage;
END_VAR
IF (currentValue > maximumValue) THEN
	THIS^.assertionWasWrong(
		message			:= message,
		additionalText	:= THIS^.getDebugInfo('valueIsMax')
	);	
END_IF
END_METHOD

(*

short summary
=================
This assertion method checks if the current value is greater than or equal to the minimum value

.. <legal notes>

legal notes
=================
| SPDX-FileCopyrightText: © 2022 ekvip automation GmbH <info@ekvip.de>
| SPDX-License-Identifier: Apache-2.0
| For details check: Apache-2.0_

.. _Apache-2.0: https://www.apache.org/licenses/LICENSE-2.0

.. </legal notes>

parameters
=================

*)

METHOD valueIsMin
VAR_INPUT
	(* current value to check *)
	currentValue	:LTIME;
	(* lower limit for the current value *)
	minimumValue	:LTIME;
	(* message if the assertion is false *)
	message			:AssertMessage;
END_VAR
IF (currentValue < minimumValue) THEN
	THIS^.assertionWasWrong(
		message			:= message,
		additionalText	:= THIS^.getDebugInfo('valueIsMin')
	);	
END_IF
END_METHOD

(*

short summary
=================
This assertion method checks if the current value is not equal to the unexpected value

.. <legal notes>

legal notes
=================
| SPDX-FileCopyrightText: © 2022 ekvip automation GmbH <info@ekvip.de>
| SPDX-License-Identifier: Apache-2.0
| For details check: Apache-2.0_

.. _Apache-2.0: https://www.apache.org/licenses/LICENSE-2.0

.. </legal notes>

parameters
=================

*)

METHOD valueIsNotEqualTo
VAR_INPUT
	(* current value to check *)
	currentValue	:LTIME;
	(* unexpected value to compare *)
	unexpectedValue	:LTIME;
	(* message if the assertion is false *)
	message			:AssertMessage;
END_VAR
IF (currentValue = unexpectedValue) THEN
	THIS^.assertionWasWrong(
		message			:= message,
		additionalText	:= THIS^.getDebugInfo('valueIsNotEqualTo')
	);	
END_IF
END_METHOD

END_FUNCTION_BLOCK

// ---- Assertor/classes/AbstractAssertor.TcPOU
(*

short summary
=================
| This abstract class provides assert statements in a `fluent interface`_ style for the most common data types. 
| It implements the interfaces :ref:`IAssertor` and :ref:`IAssertCallBack`
| If you need assertion statements you've to extend this class and you've to overwrite the methods
| :ref:`AbstractAssertor.assertionWasWrong`
| :ref:`AbstractAssertor.className`

.. _`fluent interface`: https://en.wikipedia.org/wiki/Fluent_interface

.. <legal notes>

legal notes
=================
| SPDX-FileCopyrightText: © 2022 ekvip automation GmbH <info@ekvip.de>
| SPDX-License-Identifier: Apache-2.0
| For details check: Apache-2.0_

.. _Apache-2.0: https://www.apache.org/licenses/LICENSE-2.0

.. </legal notes>

methods and properties
=======================

*)

{attribute 'reflection'}
FUNCTION_BLOCK ABSTRACT AbstractAssertor EXTENDS CNM_AbstractObject.Object IMPLEMENTS IAssertor, IAssertCallBack
VAR
	(* class to handle all the worth assertions *)
	{attribute 'hide'}
	assertions	:Assertions();
END_VAR

(*

short summary
=================
Returns the interface :ref:`IAssertions`
to get access to the assert statements

.. <legal notes>

legal notes
=================
| SPDX-FileCopyrightText: © 2022 ekvip automation GmbH <info@ekvip.de>
| SPDX-License-Identifier: Apache-2.0
| For details check: Apache-2.0_

.. _Apache-2.0: https://www.apache.org/licenses/LICENSE-2.0

.. </legal notes>

methods
==================

*)

PROPERTY assert :IAssertions
GET
assert := THIS^.assertions;
END_GET
END_PROPERTY

(*

short summary
=================
This method is called if an assertion was ``FALSE``

.. <legal notes>

legal notes
=================
| SPDX-FileCopyrightText: © 2022 ekvip automation GmbH <info@ekvip.de>
| SPDX-License-Identifier: Apache-2.0
| For details check: Apache-2.0_

.. _Apache-2.0: https://www.apache.org/licenses/LICENSE-2.0

.. </legal notes>

parameters
=================

*)

METHOD ABSTRACT assertionWasWrong
VAR_INPUT
	(* caller object of the method *)
	caller			:CNM_AbstractObject.IObject;
	(* alarm message *)
	message			:AssertMessage;
	(* debugging information *) 
	additionalText	:Tc2_System.T_MaxString;
END_VAR
END_METHOD

(*

short summary
=================
This abstract property returns the class name of the concrete object, 
It's for debugging purpose

.. attention:: 
	For derivations: **It is necessary that this property is overridden by the concrete class**

.. <legal notes>

legal notes
=================
| SPDX-FileCopyrightText: © 2022 ekvip automation GmbH <info@ekvip.de>
| SPDX-License-Identifier: Apache-2.0
| For details check: Apache-2.0_

.. _Apache-2.0: https://www.apache.org/licenses/LICENSE-2.0

.. </legal notes>

*)

PROPERTY ABSTRACT className :CNM_AbstractObject.ClassName
GET
END_GET
END_PROPERTY

(*

short summary
=================
The constructor ``FB_init`` is needed to create an unique hash code.
The hash code is a pseudo random number create with a xorshift_ algorithm.
It can be overwritten on derivations, because it will be called implicit, ``SUPER^.FB_init()`` is not required.
For more information check: `Behavoir with derived function blocks`_

.. _Behavoir with derived function blocks: https://infosys.beckhoff.com/content/1033/tc3_plc_intro/5482088715.html?id=6983869892358031022
.. _xorshift: https://en.wikipedia.org/wiki/Xorshift

.. <legal notes>

legal notes
=================
| SPDX-FileCopyrightText: © 2022 ekvip automation GmbH <info@ekvip.de>
| SPDX-License-Identifier: Apache-2.0
| For details check: Apache-2.0_

.. _Apache-2.0: https://www.apache.org/licenses/LICENSE-2.0

.. </legal notes>

parameters
=================

*)

METHOD FB_init :BOOL;
VAR_INPUT
	(* if TRUE, the retain variables are initialized (warm start / cold start)*)
	bInitRetains	:BOOL;
	(* if TRUE, the instance afterwards gets moved into the copy code (online change) *)
	bInCopyCode		:BOOL;  
END_VAR
VAR
	{attribute 'hide'}
	newHashstate3		:Hashcode;
END_VAR
VAR CONSTANT
	{attribute 'hide'}
	NUMBER_OF_LEFT_SHIFTS		:UINT	:= 17;
	{attribute 'hide'}
	NUMBER_OF_LEFT_ROTATIONS	:UINT   := 45;
END_VAR
THIS^.assertions.setCallBack(THIS^);
END_METHOD

END_FUNCTION_BLOCK

// ---- Project Information/F_GetCompany.TcPOU
// This function has been automatically generated from the project information.
{attribute 'signature_flag' := '1073741824'}
{attribute 'TcGenerated'}
{attribute 'no-analysis'}
FUNCTION F_GetCompany : WSTRING
VAR_INPUT
	
END_VAR

F_GetCompany := "ekvip automation GmbH";

END_FUNCTION

// ---- Project Information/F_GetTitle.TcPOU
// This function has been automatically generated from the project information.
{attribute 'signature_flag' := '1073741824'}
{attribute 'TcGenerated'}
{attribute 'no-analysis'}
FUNCTION F_GetTitle : WSTRING
VAR_INPUT
	
END_VAR

F_GetTitle := "CNM_AssertionInterfaceLib";

END_FUNCTION

// ---- Project Information/F_GetVersion.TcPOU
// This function has been automatically generated from the project information.
{attribute 'signature_flag' := '1073741824'}
{attribute 'TcGenerated'}
{attribute 'no-analysis'}
FUNCTION F_GetVersion : ST_LibVersion
VAR_INPUT
	
END_VAR

F_GetVersion.iMajor := 5;
F_GetVersion.iMinor := 0;
F_GetVersion.iBuild := 0;
F_GetVersion.iRevision := 0;
F_GetVersion.sVersion := '5.0.0.0';
F_GetVersion.nFlags := 0;

END_FUNCTION
